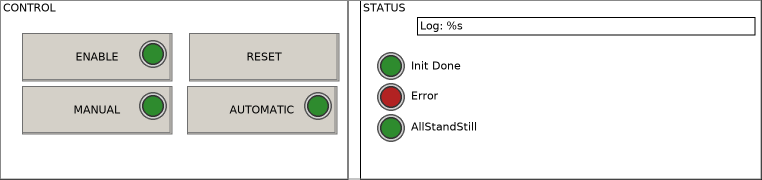
VISUALIZATION VI_XTSHomeVisu  // 762x180
VAR_IN_OUT
	xts : XTS_System;
END_VAR
    Rectangle (360,0 402x180), "STATUS"
    Rectangle (0,0 348x180), "CONTROL"
    Button (22,33 150x48), "ENABLE"
        toggle xts.bEnable
    Button (22,86 150x48), "MANUAL"
        toggle xts.bManual
    Button (187,86 150x48), "AUTOMATIC"
        toggle xts.bAutomatic
    Lamp1 (375,50 32x32), variable: xts.bInitDone, style: Lamp-Lamp1-Green
    Label (408,51 110x30), "Init Done"
    Lamp1 (137,90 32x32), variable: xts.bInManual, style: Lamp-Lamp1-Green
    Lamp1 (302,90 32x32), variable: xts.bInAutomatic, style: Lamp-Lamp1-Green
    Lamp1 (375,81 32x32), variable: xts.bError, style: Lamp-Lamp1-Red
    Label (408,81 110x30), "Error"
    Button (189,33 150x48), "RESET"
        tap xts.bReset
    Rectangle (417,17 338x18), "Log: %s", text variable: xts.sLog
        OnMouseClick: write the text variable via Default
    Lamp1 (375,112 32x32), variable: xts.bAllMoversStandStill, style: Lamp-Lamp1-Green
    Label (408,112 110x30), "AllStandStill"
    Lamp1 (137,38 32x32), variable: xts.bEnabled, style: Lamp-Lamp1-Green
END_VISUALIZATION

(* stored: Version 1.1.0.1, ProductVersion 3.1.4024.11
   Visu VI_XTSHomeVisu: Id {7519b7d6-9bdb-4064-9291-04f668dd61c0} *)
